DATA_BLOCK "CODE READING ANGLE"   // DB15
VERSION : 0.1
// stored: AutoNumber true, DBAccessibleFromOPCUA true, DBAccessibleFromWebserver true, InstanceOfName CODE READING, InstanceOfType FB
"CODE READING"
BEGIN
   scannerReading[0] := '$00';
   scannerReading[1] := ',';
   scannerReading[2] := '$00';
   scannerReading[3] := ',';
   scannerReading[4] := '$00';
   scannerReading[5] := ',';
   scannerReading[6] := '$00';
   scannerReading[7] := '4';
   scannerReading[8] := '[';
   scannerReading[9] := ')';
   scannerReading[10] := '>';
   scannerReading[11] := '0';
   scannerReading[12] := '6';
   scannerReading[13] := 'P';
   scannerReading[14] := '1';
   scannerReading[15] := '3';
   scannerReading[16..17] := '5';
   scannerReading[18] := '1';
   scannerReading[19] := '8';
   scannerReading[20] := '0';
   scannerReading[21] := '4';
   scannerReading[22] := '1';
   scannerReading[23] := '2';
   scannerReading[24] := 'V';
   scannerReading[25] := '8';
   scannerReading[26] := '1';
   scannerReading[27] := '3';
   scannerReading[28] := '1';
   scannerReading[29] := '2';
   scannerReading[30] := '0';
   scannerReading[31] := '8';
   scannerReading[32] := '2';
   scannerReading[33] := '1';
   scannerReading[34] := 'T';
   scannerReading[35] := '2';
   scannerReading[36] := '4';
   scannerReading[37] := '1';
   scannerReading[38] := '2';
   scannerReading[39] := '9';
   scannerReading[40] := 'F';
   scannerReading[41] := '3';
   scannerReading[42] := '8';
   scannerReading[43] := '7';
   scannerReading[44] := '0';
   scannerReading[45] := '4';
   scannerReading[46] := '9';
   scannerReading[47] := '4';
   scannerReading[48] := '0';
   scannerReading[49] := '1';
   scannerReading[50..51] := 'I';
   scannerReading[52] := '4';
   scannerReading[53] := 'D';
   scannerReading[54] := '0';
   scannerReading[55] := '8';
   scannerReading[56] := '7';
   scannerReading[57] := 'X';
   scannerReading[58] := 'M';
   scannerReading[59] := '$R';
   scannerReading[60..135] := '$00';
   scannerReading[136..254] := ' ';
   ScannerReadTimer.PT := T#50MS;
   ScannerReadTimer.IN := FALSE;
END_DATA_BLOCK

DATA_BLOCK "CODE READING NEST"   // DB3
VERSION : 0.1
// stored: AutoNumber true, DBAccessibleFromOPCUA true, DBAccessibleFromWebserver true, InstanceOfName CODE READING, InstanceOfType FB
"CODE READING"
BEGIN
   scannerReading[0] := '$00';
   scannerReading[1] := 'X';
   scannerReading[2] := '$00';
   scannerReading[3] := 'X';
   scannerReading[4] := '$00';
   scannerReading[5] := 'X';
   scannerReading[6] := '$00';
   scannerReading[7] := '$1E';
   scannerReading[8] := 'V';
   scannerReading[9..10] := '0';
   scannerReading[11] := '8';
   scannerReading[12] := '3';
   scannerReading[13] := '4';
   scannerReading[14] := '5';
   scannerReading[15] := 'Y';
   scannerReading[16] := '4';
   scannerReading[17] := '2';
   scannerReading[18] := '5';
   scannerReading[19] := '9';
   scannerReading[20] := '6';
   scannerReading[21] := '9';
   scannerReading[22] := '8';
   scannerReading[23] := 'X';
   scannerReading[24] := 'R';
   scannerReading[25] := '0';
   scannerReading[26..27] := '1';
   scannerReading[28] := '4';
   scannerReading[29] := '6';
   scannerReading[30] := '4';
   scannerReading[31] := '2';
   scannerReading[32] := '4';
   scannerReading[33] := '0';
   scannerReading[34] := '8';
   scannerReading[35] := '0';
   scannerReading[36] := '1';
   scannerReading[37] := '$R';
   scannerReading[38..135] := '$00';
   scannerReading[136..254] := ' ';
   ScannerReadTimer.PT := T#50MS;
   ScannerReadTimer.IN := FALSE;
END_DATA_BLOCK

DATA_BLOCK "CODE READING UPPER"   // DB12
VERSION : 0.1
// stored: AutoNumber true, DBAccessibleFromOPCUA true, DBAccessibleFromWebserver true, InstanceOfName CODE READING, InstanceOfType FB
"CODE READING"
BEGIN
   scannerReading[0] := '$00';
   scannerReading[1] := 'n';
   scannerReading[2] := '$00';
   scannerReading[3] := 'n';
   scannerReading[4] := '$00';
   scannerReading[5] := 'n';
   scannerReading[6] := '$00';
   scannerReading[7] := '$06';
   scannerReading[8] := 'E';
   scannerReading[9..10] := 'R';
   scannerReading[11] := 'O';
   scannerReading[12] := 'R';
   scannerReading[13] := '$R';
   scannerReading[14..135] := '$00';
   scannerReading[136..254] := ' ';
   ScannerReadTimer.PT := T#50MS;
   ScannerReadTimer.IN := FALSE;
END_DATA_BLOCK

DATA_BLOCK "Time System_DB"   // DB32
VERSION : 0.1
// stored: AutoNumber true, DBAccessibleFromOPCUA true, DBAccessibleFromWebserver true, InstanceOfName Time System, InstanceOfType FB
"Time System"
BEGIN
   nCycleTimeArray[0..5] := 0.0;
   tCycleTime.PT := T#0MS;
   tCycleTime.IN := FALSE;
   timesCounter.CU := FALSE;
   timesCounter.CD := FALSE;
   timesCounter.R := FALSE;
   timesCounter.LD := FALSE;
   timesCounter.QU := FALSE;
   timesCounter.QD := FALSE;
   timesCounter.PV := 5;
   timesCounter.CV := 0;
END_DATA_BLOCK
